DATA_BLOCK "Main_DB"
{ S7_Optimized_Access := 'TRUE' }
AUTHOR : 'Searinox(Gerrit_Vogtlaender)'
FAMILY : AKK
VERSION : 0.1
NON_RETAIN
"MainInstane"

BEGIN

END_DATA_BLOCK

